ABB RAPID module: RobatechData.sysx

MODULE RobatechData(SYSMODULE)
    PERS tooldata tGlueGun:=[TRUE,[[0,0,1],[1,0,0,0]],[1,[0,0,0],[1,0,0,0],0,0,0]];
ENDMODULE
